
FUNCTION CB_lt_tod : BOOL


TITLE = ' Test Whether IN0 is strictly less than IN1 '
VERSION : '1.0'
AUTHOR  : CB
NAME    : lt_tod
FAMILY  : TNI

VAR_INPUT
    IN0 : TOD;
    IN1 : TOD;
END_VAR

BEGIN

CB_lt_tod := (IN0 < IN1);

END_FUNCTION
